# EPICS substitutions: db/Beckhoff_6XXX/ecmcEL6002.substitutions
file "ecmcEcSlave.template"
{
  pattern {}
          {}
}

file "ecmcEL6002-chX.template"
{
  pattern {CH_ID, NELM }
          {1,     22   }
          {2,     22   }
}
